# EPICS autosave request: mrfApp/Db/evg-template-mxc.inc.req
$(P)$(R)MXC@MXC_NUM@:MapTo:EvTrig0.VAL
$(P)$(R)MXC@MXC_NUM@:MapTo:EvTrig1.VAL
$(P)$(R)MXC@MXC_NUM@:MapTo:EvTrig2.VAL
$(P)$(R)MXC@MXC_NUM@:MapTo:EvTrig3.VAL
$(P)$(R)MXC@MXC_NUM@:MapTo:EvTrig4.VAL
$(P)$(R)MXC@MXC_NUM@:MapTo:EvTrig5.VAL
$(P)$(R)MXC@MXC_NUM@:MapTo:EvTrig6.VAL
$(P)$(R)MXC@MXC_NUM@:MapTo:EvTrig7.VAL
$(P)$(R)MXC@MXC_NUM@:Prescaler.VAL
$(P)$(R)MXC@MXC_NUM@:ResetState.VAL
